LIN {X 0,Y 115.53,Z 526.027,A -85,B 0,C 180,E1 -30181.612,E2 -30181.612} C_VEL
LIN {X 0,Y 120.51,Z 530.093,A -85,B 0,C 180,E1 -30175.516,E2 -30175.516} C_VEL
LIN {X 0,Y 127.732,Z 533.715,A -85,B 0,C 180,E1 -30169.276,E2 -30169.276} C_VEL
LIN {X 0,Y 137.279,Z 536.546,A -85,B 0,C 180,E1 -30163.425,E2 -30163.425} C_VEL
LIN {X 0,Y 149.17,Z 538.493,A -85,B 0,C 180,E1 -30158.125,E2 -30158.125} C_VEL
LIN {X 0,Y 161.998,Z 539.441,A -85,B 0,C 180,E1 -30153.813,E2 -30153.813} C_VEL
LIN {X 0,Y 176.224,Z 539.515,A -85,B 0,C 180,E1 -30150,E2 -30150} C_VEL
LIN {X 0,Y 161.998,Z 539.441,A -85,B 0,C 180,E1 -30146.187,E2 -30146.187} C_VEL
LIN {X 0,Y 156.307,Z 539.2,A -85,B 0,C 180,E1 -30144.414,E2 -30144.414} C_VEL
LIN {X 0,Y 151.525,Z 539.005,A -85,B 0,C 180,E1 -30143.113,E2 -30143.113} C_VEL
LIN {X 0,Y 135.833,Z 538.437,A -85,B 0,C 180,E1 -30139.705,E2 -30139.705} C_VEL
LIN {X 0,Y 131.312,Z 537.898,A -85,B 0,C 180,E1 -30138.103,E2 -30138.103} C_VEL
LIN {X 0,Y 130.038,Z 537.644,A -85,B 0,C 180,E1 -30137.459,E2 -30137.459} C_VEL
LIN {X 0,Y 123.595,Z 536.121,A -85,B 0,C 180,E1 -30133.482,E2 -30133.482} C_VEL
LIN {X 0,Y 115.033,Z 532.752,A -85,B 0,C 180,E1 -30126.405,E2 -30126.405} C_VEL
LIN {X 0,Y 108.205,Z 527.615,A -85,B 0,C 180,E1 -30117.599,E2 -30117.599} C_VEL
LIN {X 0,Y 105.051,Z 522.639,A -85,B 0,C 180,E1 -30110.293,E2 -30110.293} C_VEL
LIN {X 0,Y 103.843,Z 517.611,A -85,B 0,C 180,E1 -30103.904,E2 -30103.904} C_VEL
LIN {X 0,Y 104.036,Z 511.583,A -85,B 0,C 180,E1 -30097.441,E2 -30097.441} C_VEL
LIN {X 0,Y 105.392,Z 504.732,A -85,B 0,C 180,E1 -30091.29,E2 -30091.29} C_VEL
LIN {X 0,Y 107.89,Z 496.243,A -85,B 0,C 180,E1 -30085.046,E2 -30085.046} C_VEL
LIN {X 0,Y 110.837,Z 487.656,A -85,B 0,C 180,E1 -30079.923,E2 -30079.923} C_VEL
LIN {X 0,Y 114.109,Z 478.288,A -85,B 0,C 180,E1 -30075.415,E2 -30075.415} C_VEL
LIN {X 0,Y 115.916,Z 472.807,A -85,B 0,C 180,E1 -30072.918,E2 -30072.918} C_VEL
LIN {X 0,Y 116.839,Z 468.521,A -85,B 0,C 180,E1 -30070.394,E2 -30070.394} C_VEL
LIN {X 0,Y 117.39,Z 465.488,A -85,B 0,C 180,E1 -30067.787,E2 -30067.787} C_VEL
LIN {X 0,Y 117.568,Z 464.579,A -85,B 0,C 180,E1 -30066.865,E2 -30066.865} C_VEL
LIN {X 0,Y 117.839,Z 462.307,A -85,B 0,C 180,E1 -30063.417,E2 -30063.417} C_VEL
LIN {X 0,Y 118.156,Z 460.957,A -85,B 0,C 180,E1 -30059.998,E2 -30059.998} C_VEL
LIN {X 0,Y 117.866,Z 461.826,A -85,B 0,C 180,E1 -30059.712,E2 -30059.712} C_VEL
LIN {X 0,Y 112.451,Z 474.621,A -85,B 0,C 180,E1 -30059.431,E2 -30059.431} C_VEL
LIN {X 0,Y 106.309,Z 485.523,A -85,B 0,C 180,E1 -30059.086,E2 -30059.086} C_VEL
LIN {X 0,Y 100.172,Z 494.46,A -85,B 0,C 180,E1 -30058.699,E2 -30058.699} C_VEL
LIN {X 0,Y 93.165,Z 502.98,A -85,B 0,C 180,E1 -30058.202,E2 -30058.202} C_VEL
LIN {X 0,Y 86.169,Z 510.193,A -85,B 0,C 180,E1 -30057.561,E2 -30057.561} C_VEL
LIN {X 0,Y 79.184,Z 516.388,A -85,B 0,C 180,E1 -30056.836,E2 -30056.836} C_VEL
LIN {X 0,Y 70.48,Z 522.921,A -85,B 0,C 180,E1 -30055.659,E2 -30055.659} C_VEL
LIN {X 0,Y 61.651,Z 528.476,A -85,B 0,C 180,E1 -30054.038,E2 -30054.038} C_VEL
LIN {X 0,Y 52.375,Z 533.31,A -85,B 0,C 180,E1 -30051.657,E2 -30051.657} C_VEL
LIN {X 0,Y 43.038,Z 537.243,A -85,B 0,C 180,E1 -30048.451,E2 -30048.451} C_VEL
LIN {X 0,Y 36.381,Z 539.615,A -85,B 0,C 180,E1 -30044.987,E2 -30044.987} C_VEL
LIN {X 0,Y 29.882,Z 541.418,A -85,B 0,C 180,E1 -30040.178,E2 -30040.178} C_VEL
LIN {X 0,Y 18.304,Z 543.885,A -85,B 0,C 180,E1 -30020.164,E2 -30020.164} C_VEL
LIN {X 0,Y 14.225,Z 544.486,A -85,B 0,C 180,E1 -29999.608,E2 -29999.608} C_VEL
LIN {X 0,Y 12.872,Z 544.652,A -85,B 0,C 180,E1 -29970,E2 -29970} C_VEL
LIN {X 0,Y 14.256,Z 544.487,A -85,B 0,C 180,E1 -29940.464,E2 -29940.464} C_VEL
LIN {X 0,Y 18.309,Z 543.885,A -85,B 0,C 180,E1 -29919.854,E2 -29919.854} C_VEL
LIN {X 0,Y 29.882,Z 541.418,A -85,B 0,C 180,E1 -29899.823,E2 -29899.823} C_VEL
LIN {X 0,Y 39.699,Z 538.463,A -85,B 0,C 180,E1 -29893.184,E2 -29893.184} C_VEL
LIN {X 0,Y 49.826,Z 534.472,A -85,B 0,C 180,E1 -29889.129,E2 -29889.129} C_VEL
LIN {X 0,Y 56.656,Z 531.254,A -85,B 0,C 180,E1 -29887.088,E2 -29887.088} C_VEL
LIN {X 0,Y 67.008,Z 525.231,A -85,B 0,C 180,E1 -29884.883,E2 -29884.883} C_VEL
LIN {X 0,Y 75.698,Z 519.138,A -85,B 0,C 180,E1 -29883.592,E2 -29883.592} C_VEL
LIN {X 0,Y 84.419,Z 511.817,A -85,B 0,C 180,E1 -29882.578,E2 -29882.578} C_VEL
LIN {X 0,Y 91.412,Z 504.896,A -85,B 0,C 180,E1 -29881.903,E2 -29881.903} C_VEL
LIN {X 0,Y 98.419,Z 496.726,A -85,B 0,C 180,E1 -29881.402,E2 -29881.402} C_VEL
LIN {X 0,Y 104.555,Z 488.223,A -85,B 0,C 180,E1 -29881.004,E2 -29881.004} C_VEL
LIN {X 0,Y 109.818,Z 479.515,A -85,B 0,C 180,E1 -29880.71,E2 -29880.71} C_VEL
LIN {X 0,Y 114.593,Z 469.885,A -85,B 0,C 180,E1 -29880.479,E2 -29880.479} C_VEL
LIN {X 0,Y 117.865,Z 461.832,A -85,B 0,C 180,E1 -29880.325,E2 -29880.325} C_VEL
LIN {X 0,Y 118.162,Z 460.939,A -85,B 0,C 180,E1 -29880.002,E2 -29880.002} C_VEL
LIN {X 0,Y 117.775,Z 462.852,A -85,B 0,C 180,E1 -29875.578,E2 -29875.578} C_VEL
LIN {X 0,Y 117.585,Z 464.537,A -85,B 0,C 180,E1 -29873.136,E2 -29873.136} C_VEL
LIN {X 0,Y 117.066,Z 467.337,A -85,B 0,C 180,E1 -29870.499,E2 -29870.499} C_VEL
LIN {X 0,Y 116.536,Z 470.027,A -85,B 0,C 180,E1 -29868.611,E2 -29868.611} C_VEL
LIN {X 0,Y 115.614,Z 473.856,A -85,B 0,C 180,E1 -29866.554,E2 -29866.554} C_VEL
LIN {X 0,Y 111.97,Z 484.489,A -85,B 0,C 180,E1 -29861.712,E2 -29861.712} C_VEL
LIN {X 0,Y 109.139,Z 492.578,A -85,B 0,C 180,E1 -29857.273,E2 -29857.273} C_VEL
LIN {X 0,Y 106.805,Z 499.724,A -85,B 0,C 180,E1 -29852.576,E2 -29852.576} C_VEL
LIN {X 0,Y 104.762,Z 507.268,A -85,B 0,C 180,E1 -29846.586,E2 -29846.586} C_VEL
LIN {X 0,Y 103.737,Z 514.599,A -85,B 0,C 180,E1 -29839.467,E2 -29839.467} C_VEL
LIN {X 0,Y 104.4,Z 520.737,A -85,B 0,C 180,E1 -29832.229,E2 -29832.229} C_VEL
LIN {X 0,Y 106.954,Z 526.067,A -85,B 0,C 180,E1 -29824.784,E2 -29824.784} C_VEL
LIN {X 0,Y 111.232,Z 530.386,A -85,B 0,C 180,E1 -29817.806,E2 -29817.806} C_VEL
LIN {X 0,Y 117.751,Z 534.005,A -85,B 0,C 180,E1 -29810.984,E2 -29810.984} C_VEL
LIN {X 0,Y 124.29,Z 536.317,A -85,B 0,C 180,E1 -29806.005,E2 -29806.005} C_VEL
LIN {X 0,Y 135.51,Z 538.538,A -85,B 0,C 180,E1 -29799.812,E2 -29799.812} C_VEL
LIN {X 0,Y 148.1,Z 539.687,A -85,B 0,C 180,E1 -29794.785,E2 -29794.785} C_VEL
LIN {X 0,Y 164.311,Z 539.834,A -85,B 0,C 180,E1 -29790,E2 -29790} C_VEL
LIN {X 0,Y 148.1,Z 539.687,A -85,B 0,C 180,E1 -29785.215,E2 -29785.215} C_VEL
LIN {X 0,Y 135.51,Z 538.538,A -85,B 0,C 180,E1 -29780.188,E2 -29780.188} C_VEL
LIN {X 0,Y 130.038,Z 537.644,A -85,B 0,C 180,E1 -29777.459,E2 -29777.459} C_VEL
LIN {X 0,Y 125.995,Z 536.984,A -85,B 0,C 180,E1 -29775.552,E2 -29775.552} C_VEL
LIN {X 0,Y 112.333,Z 535.461,A -85,B 0,C 180,E1 -29770.066,E2 -29770.066} C_VEL
LIN {X 0,Y 108.732,Z 534.57,A -85,B 0,C 180,E1 -29767.694,E2 -29767.694} C_VEL
LIN {X 0,Y 107.819,Z 534.193,A -85,B 0,C 180,E1 -29766.796,E2 -29766.796} C_VEL
LIN {X 0,Y 102.19,Z 530.522,A -85,B 0,C 180,E1 -29759.259,E2 -29759.259} C_VEL
LIN {X 0,Y 98.44,Z 525.194,A -85,B 0,C 180,E1 -29750.02,E2 -29750.02} C_VEL
LIN {X 0,Y 97.559,Z 518.271,A -85,B 0,C 180,E1 -29740.414,E2 -29740.414} C_VEL
LIN {X 0,Y 98.89,Z 511.152,A -85,B 0,C 180,E1 -29732.537,E2 -29732.537} C_VEL
LIN {X 0,Y 101.524,Z 503.604,A -85,B 0,C 180,E1 -29725.854,E2 -29725.854} C_VEL
LIN {X 0,Y 104.848,Z 495.671,A -85,B 0,C 180,E1 -29720.215,E2 -29720.215} C_VEL
LIN {X 0,Y 108.168,Z 488.054,A -85,B 0,C 180,E1 -29715.776,E2 -29715.776} C_VEL
LIN {X 0,Y 111.823,Z 479.417,A -85,B 0,C 180,E1 -29711.676,E2 -29711.676} C_VEL
LIN {X 0,Y 113.231,Z 475.646,A -85,B 0,C 180,E1 -29709.754,E2 -29709.754} C_VEL
LIN {X 0,Y 114.361,Z 471.98,A -85,B 0,C 180,E1 -29707.058,E2 -29707.058} C_VEL
LIN {X 0,Y 114.739,Z 470.338,A -85,B 0,C 180,E1 -29705.27,E2 -29705.27} C_VEL
LIN {X 0,Y 115.032,Z 469.144,A -85,B 0,C 180,E1 -29703.501,E2 -29703.501} C_VEL
LIN {X 0,Y 114.177,Z 471.006,A -85,B 0,C 180,E1 -29703.048,E2 -29703.048} C_VEL
LIN {X 0,Y 108.194,Z 482.562,A -85,B 0,C 180,E1 -29702.924,E2 -29702.924} C_VEL
LIN {X 0,Y 101.146,Z 493.131,A -85,B 0,C 180,E1 -29702.797,E2 -29702.797} C_VEL
LIN {X 0,Y 94.976,Z 500.868,A -85,B 0,C 180,E1 -29702.633,E2 -29702.633} C_VEL
LIN {X 0,Y 86.16,Z 509.999,A -85,B 0,C 180,E1 -29702.297,E2 -29702.297} C_VEL
LIN {X 0,Y 79.111,Z 516.194,A -85,B 0,C 180,E1 -29701.987,E2 -29701.987} C_VEL
LIN {X 0,Y 70.301,Z 522.727,A -85,B 0,C 180,E1 -29701.455,E2 -29701.455} C_VEL
LIN {X 0,Y 63.258,Z 527.227,A -85,B 0,C 180,E1 -29700.888,E2 -29700.888} C_VEL
LIN {X 0,Y 53.476,Z 532.382,A -85,B 0,C 180,E1 -29699.749,E2 -29699.749} C_VEL
LIN {X 0,Y 45.696,Z 535.808,A -85,B 0,C 180,E1 -29698.546,E2 -29698.546} C_VEL
LIN {X 0,Y 35.215,Z 539.42,A -85,B 0,C 180,E1 -29696.245,E2 -29696.245} C_VEL
LIN {X 0,Y 28.272,Z 541.223,A -85,B 0,C 180,E1 -29693.889,E2 -29693.889} C_VEL
LIN {X 0,Y 14.789,Z 543.69,A -85,B 0,C 180,E1 -29681.885,E2 -29681.885} C_VEL
LIN {X 0,Y 8.78,Z 544.292,A -85,B 0,C 180,E1 -29663.168,E2 -29663.168} C_VEL
LIN {X 0,Y 5.758,Z 544.457,A -85,B 0,C 180,E1 -29610,E2 -29610} C_VEL
LIN {X 0,Y 8.798,Z 544.293,A -85,B 0,C 180,E1 -29556.985,E2 -29556.985} C_VEL
LIN {X 0,Y 14.791,Z 543.691,A -85,B 0,C 180,E1 -29538.137,E2 -29538.137} C_VEL
LIN {X 0,Y 28.272,Z 541.223,A -85,B 0,C 180,E1 -29526.112,E2 -29526.112} C_VEL
LIN {X 0,Y 38.7,Z 538.268,A -85,B 0,C 180,E1 -29522.835,E2 -29522.835} C_VEL
LIN {X 0,Y 49.201,Z 534.277,A -85,B 0,C 180,E1 -29520.889,E2 -29520.889} C_VEL
LIN {X 0,Y 56.223,Z 531.059,A -85,B 0,C 180,E1 -29519.85,E2 -29519.85} C_VEL
LIN {X 0,Y 66.779,Z 525.037,A -85,B 0,C 180,E1 -29518.794,E2 -29518.794} C_VEL
LIN {X 0,Y 75.587,Z 518.944,A -85,B 0,C 180,E1 -29518.192,E2 -29518.192} C_VEL
LIN {X 0,Y 84.4,Z 511.622,A -85,B 0,C 180,E1 -29517.738,E2 -29517.738} C_VEL
LIN {X 0,Y 91.452,Z 504.701,A -85,B 0,C 180,E1 -29517.449,E2 -29517.449} C_VEL
LIN {X 0,Y 98.501,Z 496.532,A -85,B 0,C 180,E1 -29517.275,E2 -29517.275} C_VEL
LIN {X 0,Y 104.672,Z 488.029,A -85,B 0,C 180,E1 -29517.113,E2 -29517.113} C_VEL
LIN {X 0,Y 109.959,Z 479.321,A -85,B 0,C 180,E1 -29517.01,E2 -29517.01} C_VEL
LIN {X 0,Y 114.36,Z 470.588,A -85,B 0,C 180,E1 -29516.941,E2 -29516.941} C_VEL
LIN {X 0,Y 115.039,Z 469.127,A -85,B 0,C 180,E1 -29516.499,E2 -29516.499} C_VEL
LIN {X 0,Y 114.766,Z 470.276,A -85,B 0,C 180,E1 -29514.732,E2 -29514.732} C_VEL
LIN {X 0,Y 114.116,Z 472.975,A -85,B 0,C 180,E1 -29512.101,E2 -29512.101} C_VEL
LIN {X 0,Y 113.218,Z 475.674,A -85,B 0,C 180,E1 -29510.238,E2 -29510.238} C_VEL
LIN {X 0,Y 111.827,Z 479.404,A -85,B 0,C 180,E1 -29508.331,E2 -29508.331} C_VEL
LIN {X 0,Y 107.548,Z 489.598,A -85,B 0,C 180,E1 -29503.396,E2 -29503.396} C_VEL
LIN {X 0,Y 103.013,Z 500.012,A -85,B 0,C 180,E1 -29496.906,E2 -29496.906} C_VEL
LIN {X 0,Y 99.623,Z 508.727,A -85,B 0,C 180,E1 -29489.784,E2 -29489.784} C_VEL
LIN {X 0,Y 97.978,Z 514.853,A -85,B 0,C 180,E1 -29483.581,E2 -29483.581} C_VEL
LIN {X 0,Y 97.475,Z 520.931,A -85,B 0,C 180,E1 -29476.136,E2 -29476.136} C_VEL
LIN {X 0,Y 98.796,Z 526.081,A -85,B 0,C 180,E1 -29468.513,E2 -29468.513} C_VEL
LIN {X 0,Y 102.139,Z 530.53,A -85,B 0,C 180,E1 -29460.749,E2 -29460.749} C_VEL
LIN {X 0,Y 108.005,Z 534.292,A -85,B 0,C 180,E1 -29452.98,E2 -29452.98} C_VEL
LIN {X 0,Y 113.262,Z 536.417,A -85,B 0,C 180,E1 -29448.074,E2 -29448.074} C_VEL
LIN {X 0,Y 122.132,Z 538.533,A -85,B 0,C 180,E1 -29441.981,E2 -29441.981} C_VEL
LIN {X 0,Y 134.521,Z 539.916,A -85,B 0,C 180,E1 -29435.998,E2 -29435.998} C_VEL
LIN {X 0,Y 147.626,Z 540.282,A -85,B 0,C 180,E1 -29431.378,E2 -29431.378} C_VEL
LIN {X 0,Y 152.405,Z 540.153,A -85,B 0,C 180,E1 -29430,E2 -29430} C_VEL
LIN {X 0,Y 140.832,Z 540.169,A -85,B 0,C 180,E1 -29426.413,E2 -29426.413} C_VEL
LIN {X 0,Y 128.022,Z 539.297,A -85,B 0,C 180,E1 -29421.157,E2 -29421.157} C_VEL
LIN {X 0,Y 119.45,Z 537.971,A -85,B 0,C 180,E1 -29416.388,E2 -29416.388} C_VEL
LIN {X 0,Y 111.734,Z 535.891,A -85,B 0,C 180,E1 -29410.64,E2 -29410.64} C_VEL
LIN {X 0,Y 107.819,Z 534.193,A -85,B 0,C 180,E1 -29406.796,E2 -29406.796} C_VEL
LIN {X 0,Y 104.89,Z 533.159,A -85,B 0,C 180,E1 -29404.087,E2 -29404.087} C_VEL
LIN {X 0,Y 94.721,Z 530.474,A -85,B 0,C 180,E1 -29395.798,E2 -29395.798} C_VEL
LIN {X 0,Y 92.539,Z 529.043,A -85,B 0,C 180,E1 -29392.569,E2 -29392.569} C_VEL
LIN {X 0,Y 92.134,Z 528.439,A -85,B 0,C 180,E1 -29391.437,E2 -29391.437} C_VEL
LIN {X 0,Y 91.087,Z 524.144,A -85,B 0,C 180,E1 -29383.977,E2 -29383.977} C_VEL
LIN {X 0,Y 91.954,Z 517.723,A -85,B 0,C 180,E1 -29374.969,E2 -29374.969} C_VEL
LIN {X 0,Y 94.409,Z 511.216,A -85,B 0,C 180,E1 -29367.722,E2 -29367.722} C_VEL
LIN {X 0,Y 97.995,Z 503.845,A -85,B 0,C 180,E1 -29361.202,E2 -29361.202} C_VEL
LIN {X 0,Y 102.179,Z 495.907,A -85,B 0,C 180,E1 -29355.654,E2 -29355.654} C_VEL
LIN {X 0,Y 106.153,Z 488.365,A -85,B 0,C 180,E1 -29351.454,E2 -29351.454} C_VEL
LIN {X 0,Y 109.817,Z 480.976,A -85,B 0,C 180,E1 -29347.881,E2 -29347.881} C_VEL
LIN {X 0,Y 110.214,Z 480.011,A -85,B 0,C 180,E1 -29347.325,E2 -29347.325} C_VEL
LIN {X 0,Y 109.156,Z 481.709,A -85,B 0,C 180,E1 -29346.66,E2 -29346.66} C_VEL
LIN {X 0,Y 101.739,Z 492.937,A -85,B 0,C 180,E1 -29346.793,E2 -29346.793} C_VEL
LIN {X 0,Y 95.565,Z 500.675,A -85,B 0,C 180,E1 -29346.885,E2 -29346.885} C_VEL
LIN {X 0,Y 86.738,Z 509.804,A -85,B 0,C 180,E1 -29347.004,E2 -29347.004} C_VEL
LIN {X 0,Y 79.677,Z 515.999,A -85,B 0,C 180,E1 -29347.118,E2 -29347.118} C_VEL
LIN {X 0,Y 70.843,Z 522.532,A -85,B 0,C 180,E1 -29347.237,E2 -29347.237} C_VEL
LIN {X 0,Y 63.769,Z 527.032,A -85,B 0,C 180,E1 -29347.31,E2 -29347.31} C_VEL
LIN {X 0,Y 52.924,Z 532.625,A -85,B 0,C 180,E1 -29347.375,E2 -29347.375} C_VEL
LIN {X 0,Y 42.541,Z 536.854,A -85,B 0,C 180,E1 -29347.601,E2 -29347.601} C_VEL
LIN {X 0,Y 35.467,Z 539.226,A -85,B 0,C 180,E1 -29347.798,E2 -29347.798} C_VEL
LIN {X 0,Y 28.41,Z 541.029,A -85,B 0,C 180,E1 -29348.313,E2 -29348.313} C_VEL
LIN {X 0,Y 14.284,Z 543.495,A -85,B 0,C 180,E1 -29350.265,E2 -29350.265} C_VEL
LIN {X 0,Y 7.271,Z 544.097,A -85,B 0,C 180,E1 -29354.864,E2 -29354.864} C_VEL
LIN {X 0,Y 1.342,Z 544.264,A -85,B 0,C 180,E1 -29430,E2 -29430} C_VEL
LIN {X 0,Y 7.264,Z 544.098,A -85,B 0,C 180,E1 -29505.336,E2 -29505.336} C_VEL
LIN {X 0,Y 14.283,Z 543.496,A -85,B 0,C 180,E1 -29509.757,E2 -29509.757} C_VEL
LIN {X 0,Y 28.41,Z 541.029,A -85,B 0,C 180,E1 -29511.687,E2 -29511.687} C_VEL
LIN {X 0,Y 39.006,Z 538.072,A -85,B 0,C 180,E1 -29512.286,E2 -29512.286} C_VEL
LIN {X 0,Y 49.607,Z 534.082,A -85,B 0,C 180,E1 -29512.609,E2 -29512.609} C_VEL
LIN {X 0,Y 60.238,Z 528.947,A -85,B 0,C 180,E1 -29512.604,E2 -29512.604} C_VEL
LIN {X 0,Y 69.074,Z 523.687,A -85,B 0,C 180,E1 -29512.749,E2 -29512.749} C_VEL
LIN {X 0,Y 77.911,Z 517.374,A -85,B 0,C 180,E1 -29512.853,E2 -29512.853} C_VEL
LIN {X 0,Y 84.979,Z 511.428,A -85,B 0,C 180,E1 -29512.934,E2 -29512.934} C_VEL
LIN {X 0,Y 92.043,Z 504.507,A -85,B 0,C 180,E1 -29513.026,E2 -29513.026} C_VEL
LIN {X 0,Y 99.092,Z 496.338,A -85,B 0,C 180,E1 -29513.173,E2 -29513.173} C_VEL
LIN {X 0,Y 105.269,Z 487.835,A -85,B 0,C 180,E1 -29513.25,E2 -29513.25} C_VEL
LIN {X 0,Y 109.166,Z 481.695,A -85,B 0,C 180,E1 -29513.327,E2 -29513.327} C_VEL
LIN {X 0,Y 110.222,Z 479.996,A -85,B 0,C 180,E1 -29512.676,E2 -29512.676} C_VEL
LIN {X 0,Y 108.059,Z 484.613,A -85,B 0,C 180,E1 -29510.371,E2 -29510.371} C_VEL
LIN {X 0,Y 103.854,Z 492.82,A -85,B 0,C 180,E1 -29506.176,E2 -29506.176} C_VEL
LIN {X 0,Y 99.128,Z 501.682,A -85,B 0,C 180,E1 -29500.436,E2 -29500.436} C_VEL
LIN {X 0,Y 95.443,Z 508.971,A -85,B 0,C 180,E1 -29494.419,E2 -29494.419} C_VEL
LIN {X 0,Y 92.738,Z 515.274,A -85,B 0,C 180,E1 -29487.965,E2 -29487.965} C_VEL
LIN {X 0,Y 91.17,Z 521.19,A -85,B 0,C 180,E1 -29480.43,E2 -29480.43} C_VEL
LIN {X 0,Y 91.33,Z 526.254,A -85,B 0,C 180,E1 -29472.501,E2 -29472.501} C_VEL
LIN {X 0,Y 93.531,Z 530.627,A -85,B 0,C 180,E1 -29464.258,E2 -29464.258} C_VEL
LIN {X 0,Y 98.459,Z 534.578,A -85,B 0,C 180,E1 -29455.358,E2 -29455.358} C_VEL
LIN {X 0,Y 104.092,Z 536.965,A -85,B 0,C 180,E1 -29449.057,E2 -29449.057} C_VEL
LIN {X 0,Y 114.583,Z 539.286,A -85,B 0,C 180,E1 -29441.088,E2 -29441.088} C_VEL
LIN {X 0,Y 123.077,Z 540.226,A -85,B 0,C 180,E1 -29436.558,E2 -29436.558} C_VEL
LIN {X 0,Y 133.634,Z 540.627,A -85,B 0,C 180,E1 -29432.281,E2 -29432.281} C_VEL
LIN {X 0,Y 140.49,Z 540.472,A -85,B 0,C 180,E1 -29430,E2 -29430} C_VEL
LIN {X 0,Y 131.511,Z 540.565,A -85,B 0,C 180,E1 -29426.937,E2 -29426.937} C_VEL
LIN {X 0,Y 120.584,Z 540.045,A -85,B 0,C 180,E1 -29422.211,E2 -29422.211} C_VEL
LIN {X 0,Y 108.962,Z 538.266,A -85,B 0,C 180,E1 -29415.049,E2 -29415.049} C_VEL
LIN {X 0,Y 101.541,Z 535.979,A -85,B 0,C 180,E1 -29408.287,E2 -29408.287} C_VEL
LIN {X 0,Y 94.891,Z 532.04,A -85,B 0,C 180,E1 -29398.773,E2 -29398.773} C_VEL
LIN {X 0,Y 92.134,Z 528.439,A -85,B 0,C 180,E1 -29391.437,E2 -29391.437} C_VEL
LIN {X 0,Y 90.803,Z 526.757,A -85,B 0,C 180,E1 -29387.988,E2 -29387.988} C_VEL
LIN {X 0,Y 86.123,Z 522.502,A -85,B 0,C 180,E1 -29377.176,E2 -29377.176} C_VEL
LIN {X 0,Y 85.979,Z 520.542,A -85,B 0,C 180,E1 -29373.482,E2 -29373.482} C_VEL
LIN {X 0,Y 86.244,Z 519.758,A -85,B 0,C 180,E1 -29372.297,E2 -29372.297} C_VEL
LIN {X 0,Y 89.862,Z 512.848,A -85,B 0,C 180,E1 -29364.119,E2 -29364.119} C_VEL
LIN {X 0,Y 94.345,Z 505.462,A -85,B 0,C 180,E1 -29357.333,E2 -29357.333} C_VEL
LIN {X 0,Y 99.444,Z 497.412,A -85,B 0,C 180,E1 -29351.699,E2 -29351.699} C_VEL
LIN {X 0,Y 100.186,Z 496.144,A -85,B 0,C 180,E1 -29350.867,E2 -29350.867} C_VEL
LIN {X 0,Y 93.168,Z 504.314,A -85,B 0,C 180,E1 -29351.302,E2 -29351.302} C_VEL
LIN {X 0,Y 84.371,Z 512.861,A -85,B 0,C 180,E1 -29351.837,E2 -29351.837} C_VEL
LIN {X 0,Y 73.841,Z 521.183,A -85,B 0,C 180,E1 -29352.697,E2 -29352.697} C_VEL
LIN {X 0,Y 65.059,Z 526.838,A -85,B 0,C 180,E1 -29353.54,E2 -29353.54} C_VEL
LIN {X 0,Y 55.435,Z 531.927,A -85,B 0,C 180,E1 -29354.684,E2 -29354.684} C_VEL
LIN {X 0,Y 47.515,Z 535.42,A -85,B 0,C 180,E1 -29355.97,E2 -29355.97} C_VEL
LIN {X 0,Y 37.116,Z 539.031,A -85,B 0,C 180,E1 -29358.783,E2 -29358.783} C_VEL
LIN {X 0,Y 23.544,Z 542.23,A -85,B 0,C 180,E1 -29366.427,E2 -29366.427} C_VEL
LIN {X 0,Y 17.068,Z 543.301,A -85,B 0,C 180,E1 -29374.56,E2 -29374.56} C_VEL
LIN {X 0,Y 11.406,Z 543.903,A -85,B 0,C 180,E1 -29391.966,E2 -29391.966} C_VEL
LIN {X 0,Y 8.433,Z 544.07,A -85,B 0,C 180,E1 -29430,E2 -29430} C_VEL
LIN {X 0,Y 11.389,Z 543.903,A -85,B 0,C 180,E1 -29468.101,E2 -29468.101} C_VEL
LIN {X 0,Y 17.065,Z 543.301,A -85,B 0,C 180,E1 -29485.452,E2 -29485.452} C_VEL
LIN {X 0,Y 30.268,Z 540.835,A -85,B 0,C 180,E1 -29498.242,E2 -29498.242} C_VEL
LIN {X 0,Y 40.587,Z 537.877,A -85,B 0,C 180,E1 -29502.242,E2 -29502.242} C_VEL
LIN {X 0,Y 47.518,Z 535.419,A -85,B 0,C 180,E1 -29504.016,E2 -29504.016} C_VEL
LIN {X 0,Y 58.043,Z 530.669,A -85,B 0,C 180,E1 -29505.612,E2 -29505.612} C_VEL
LIN {X 0,Y 68.572,Z 524.648,A -85,B 0,C 180,E1 -29506.816,E2 -29506.816} C_VEL
LIN {X 0,Y 77.355,Z 518.555,A -85,B 0,C 180,E1 -29507.595,E2 -29507.595} C_VEL
LIN {X 0,Y 84.384,Z 512.859,A -85,B 0,C 180,E1 -29508.121,E2 -29508.121} C_VEL
LIN {X 0,Y 93.172,Z 504.314,A -85,B 0,C 180,E1 -29508.688,E2 -29508.688} C_VEL
LIN {X 0,Y 100.183,Z 496.145,A -85,B 0,C 180,E1 -29509.142,E2 -29509.142} C_VEL
LIN {X 0,Y 94.35,Z 505.456,A -85,B 0,C 180,E1 -29502.668,E2 -29502.668} C_VEL
LIN {X 0,Y 89.038,Z 514.197,A -85,B 0,C 180,E1 -29494.522,E2 -29494.522} C_VEL
LIN {X 0,Y 85.528,Z 521.444,A -85,B 0,C 180,E1 -29485.255,E2 -29485.255} C_VEL
LIN {X 0,Y 84.543,Z 525.778,A -85,B 0,C 180,E1 -29478.318,E2 -29478.318} C_VEL
LIN {X 0,Y 85.383,Z 530.66,A -85,B 0,C 180,E1 -29468.568,E2 -29468.568} C_VEL
LIN {X 0,Y 89.317,Z 534.857,A -85,B 0,C 180,E1 -29458.171,E2 -29458.171} C_VEL
LIN {X 0,Y 93.455,Z 536.993,A -85,B 0,C 180,E1 -29452.086,E2 -29452.086} C_VEL
LIN {X 0,Y 101.464,Z 539.209,A -85,B 0,C 180,E1 -29444.145,E2 -29444.145} C_VEL
LIN {X 0,Y 113.189,Z 540.585,A -85,B 0,C 180,E1 -29436.579,E2 -29436.579} C_VEL
LIN {X 0,Y 126.513,Z 540.847,A -85,B 0,C 180,E1 -29430.819,E2 -29430.819} C_VEL
LIN {X 0,Y 128.847,Z 540.784,A -85,B 0,C 180,E1 -29430,E2 -29430} C_VEL
LIN {X 0,Y 119.694,Z 540.864,A -85,B 0,C 180,E1 -29426.511,E2 -29426.511} C_VEL
LIN {X 0,Y 107.081,Z 540.017,A -85,B 0,C 180,E1 -29419.881,E2 -29419.881} C_VEL
LIN {X 0,Y 98.692,Z 538.557,A -85,B 0,C 180,E1 -29413.451,E2 -29413.451} C_VEL
LIN {X 0,Y 92.191,Z 536.396,A -85,B 0,C 180,E1 -29406.171,E2 -29406.171} C_VEL
LIN {X 0,Y 86.478,Z 532.314,A -85,B 0,C 180,E1 -29395.329,E2 -29395.329} C_VEL
LIN {X 0,Y 84.543,Z 527.478,A -85,B 0,C 180,E1 -29384.955,E2 -29384.955} C_VEL
LIN {X 0,Y 85.554,Z 521.443,A -85,B 0,C 180,E1 -29374.77,E2 -29374.77} C_VEL
LIN {X 0,Y 86.244,Z 519.758,A -85,B 0,C 180,E1 -29372.297,E2 -29372.297} C_VEL
LIN {X 0,Y 86.504,Z 518.36,A -85,B 0,C 180,E1 -29369.819,E2 -29369.819} C_VEL
LIN {X 0,Y 85.647,Z 514.934,A -85,B 0,C 180,E1 -29361.146,E2 -29361.146} C_VEL
LIN {X 0,Y 86.48,Z 513.232,A -85,B 0,C 180,E1 -29358.816,E2 -29358.816} C_VEL
LIN {X 0,Y 88.038,Z 511.023,A -85,B 0,C 180,E1 -29356.68,E2 -29356.68} C_VEL
LIN {X 0,Y 87.861,Z 511.04,A -85,B 0,C 180,E1 -29356.289,E2 -29356.289} C_VEL
LIN {X 0,Y 80.923,Z 516.986,A -85,B 0,C 180,E1 -29357.196,E2 -29357.196} C_VEL
LIN {X 0,Y 72.271,Z 523.298,A -85,B 0,C 180,E1 -29358.537,E2 -29358.537} C_VEL
LIN {X 0,Y 63.64,Z 528.559,A -85,B 0,C 180,E1 -29360.171,E2 -29360.171} C_VEL
LIN {X 0,Y 53.357,Z 533.692,A -85,B 0,C 180,E1 -29362.78,E2 -29362.78} C_VEL
LIN {X 0,Y 43.299,Z 537.683,A -85,B 0,C 180,E1 -29366.784,E2 -29366.784} C_VEL
LIN {X 0,Y 33.56,Z 540.64,A -85,B 0,C 180,E1 -29373.107,E2 -29373.107} C_VEL
LIN {X 0,Y 21.912,Z 543.106,A -85,B 0,C 180,E1 -29390.1,E2 -29390.1} C_VEL
LIN {X 0,Y 17.562,Z 543.708,A -85,B 0,C 180,E1 -29406.411,E2 -29406.411} C_VEL
LIN {X 0,Y 15.543,Z 543.876,A -85,B 0,C 180,E1 -29430,E2 -29430} C_VEL
LIN {X 0,Y 17.546,Z 543.709,A -85,B 0,C 180,E1 -29453.612,E2 -29453.612} C_VEL
LIN {X 0,Y 21.909,Z 543.106,A -85,B 0,C 180,E1 -29469.906,E2 -29469.906} C_VEL
LIN {X 0,Y 33.56,Z 540.64,A -85,B 0,C 180,E1 -29486.893,E2 -29486.893} C_VEL
LIN {X 0,Y 43.299,Z 537.682,A -85,B 0,C 180,E1 -29493.214,E2 -29493.214} C_VEL
LIN {X 0,Y 53.37,Z 533.691,A -85,B 0,C 180,E1 -29497.185,E2 -29497.185} C_VEL
LIN {X 0,Y 63.662,Z 528.557,A -85,B 0,C 180,E1 -29499.774,E2 -29499.774} C_VEL
LIN {X 0,Y 72.271,Z 523.298,A -85,B 0,C 180,E1 -29501.463,E2 -29501.463} C_VEL
LIN {X 0,Y 80.924,Z 516.986,A -85,B 0,C 180,E1 -29502.802,E2 -29502.802} C_VEL
LIN {X 0,Y 87.87,Z 511.04,A -85,B 0,C 180,E1 -29503.69,E2 -29503.69} C_VEL
LIN {X 0,Y 88.029,Z 511.024,A -85,B 0,C 180,E1 -29503.341,E2 -29503.341} C_VEL
LIN {X 0,Y 82.509,Z 518.748,A -85,B 0,C 180,E1 -29494.796,E2 -29494.796} C_VEL
LIN {X 0,Y 78.592,Z 525.98,A -85,B 0,C 180,E1 -29483.591,E2 -29483.591} C_VEL
LIN {X 0,Y 77.931,Z 530.624,A -85,B 0,C 180,E1 -29473.829,E2 -29473.829} C_VEL
LIN {X 0,Y 80.624,Z 535.131,A -85,B 0,C 180,E1 -29461.534,E2 -29461.534} C_VEL
LIN {X 0,Y 84.522,Z 537.492,A -85,B 0,C 180,E1 -29453.851,E2 -29453.851} C_VEL
LIN {X 0,Y 94.36,Z 540.004,A -85,B 0,C 180,E1 -29442.911,E2 -29442.911} C_VEL
LIN {X 0,Y 101.12,Z 540.83,A -85,B 0,C 180,E1 -29437.99,E2 -29437.99} C_VEL
LIN {X 0,Y 112.511,Z 541.23,A -85,B 0,C 180,E1 -29431.978,E2 -29431.978} C_VEL
LIN {X 0,Y 117.33,Z 541.096,A -85,B 0,C 180,E1 -29430,E2 -29430} C_VEL
LIN {X 0,Y 105.857,Z 541.051,A -85,B 0,C 180,E1 -29424.766,E2 -29424.766} C_VEL
LIN {X 0,Y 99.612,Z 540.73,A -85,B 0,C 180,E1 -29421.007,E2 -29421.007} C_VEL
LIN {X 0,Y 88.709,Z 538.843,A -85,B 0,C 180,E1 -29411.525,E2 -29411.525} C_VEL
LIN {X 0,Y 84.099,Z 537.271,A -85,B 0,C 180,E1 -29405.302,E2 -29405.302} C_VEL
LIN {X 0,Y 78.999,Z 533.346,A -85,B 0,C 180,E1 -29393.189,E2 -29393.189} C_VEL
LIN {X 0,Y 77.995,Z 528.409,A -85,B 0,C 180,E1 -29381.382,E2 -29381.382} C_VEL
LIN {X 0,Y 79.749,Z 523.317,A -85,B 0,C 180,E1 -29371.918,E2 -29371.918} C_VEL
LIN {X 0,Y 82.508,Z 518.749,A -85,B 0,C 180,E1 -29365.205,E2 -29365.205} C_VEL
LIN {X 0,Y 86.48,Z 513.232,A -85,B 0,C 180,E1 -29358.816,E2 -29358.816} C_VEL
LIN {X 0,Y 85.976,Z 513.469,A -85,B 0,C 180,E1 -29358.3,E2 -29358.3} C_VEL
LIN {X 0,Y 83.959,Z 514.972,A -85,B 0,C 180,E1 -29358.08,E2 -29358.08} C_VEL
LIN {X 0,Y 80.115,Z 518.157,A -85,B 0,C 180,E1 -29358.889,E2 -29358.889} C_VEL
LIN {X 0,Y 70.926,Z 525.373,A -85,B 0,C 180,E1 -29363.308,E2 -29363.308} C_VEL
LIN {X 0,Y 64.57,Z 529.46,A -85,B 0,C 180,E1 -29366.406,E2 -29366.406} C_VEL
LIN {X 0,Y 62.262,Z 530.713,A -85,B 0,C 180,E1 -29367.276,E2 -29367.276} C_VEL
LIN {X 0,Y 53.246,Z 535.03,A -85,B 0,C 180,E1 -29370.915,E2 -29370.915} C_VEL
LIN {X 0,Y 43.861,Z 538.641,A -85,B 0,C 180,E1 -29376.759,E2 -29376.759} C_VEL
LIN {X 0,Y 37.933,Z 540.445,A -85,B 0,C 180,E1 -29382.177,E2 -29382.177} C_VEL
LIN {X 0,Y 27.754,Z 542.911,A -85,B 0,C 180,E1 -29399.573,E2 -29399.573} C_VEL
LIN {X 0,Y 24.268,Z 543.514,A -85,B 0,C 180,E1 -29413.167,E2 -29413.167} C_VEL
LIN {X 0,Y 22.642,Z 543.682,A -85,B 0,C 180,E1 -29430,E2 -29430} C_VEL
LIN {X 0,Y 24.254,Z 543.514,A -85,B 0,C 180,E1 -29446.844,E2 -29446.844} C_VEL
LIN {X 0,Y 27.751,Z 542.911,A -85,B 0,C 180,E1 -29460.43,E2 -29460.43} C_VEL
LIN {X 0,Y 37.933,Z 540.445,A -85,B 0,C 180,E1 -29477.823,E2 -29477.823} C_VEL
LIN {X 0,Y 46.943,Z 537.488,A -85,B 0,C 180,E1 -29485.427,E2 -29485.427} C_VEL
LIN {X 0,Y 56.524,Z 533.496,A -85,B 0,C 180,E1 -29490.497,E2 -29490.497} C_VEL
LIN {X 0,Y 66.466,Z 528.363,A -85,B 0,C 180,E1 -29493.994,E2 -29493.994} C_VEL
LIN {X 0,Y 74.837,Z 523.104,A -85,B 0,C 180,E1 -29496.292,E2 -29496.292} C_VEL
LIN {X 0,Y 76.575,Z 521.945,A -85,B 0,C 180,E1 -29496.602,E2 -29496.602} C_VEL
LIN {X 0,Y 72.486,Z 527.747,A -85,B 0,C 180,E1 -29486.313,E2 -29486.313} C_VEL
LIN {X 0,Y 71.149,Z 531.942,A -85,B 0,C 180,E1 -29476.26,E2 -29476.26} C_VEL
LIN {X 0,Y 72.327,Z 535.403,A -85,B 0,C 180,E1 -29465.662,E2 -29465.662} C_VEL
LIN {X 0,Y 74.898,Z 537.551,A -85,B 0,C 180,E1 -29457.98,E2 -29457.98} C_VEL
LIN {X 0,Y 81.196,Z 539.778,A -85,B 0,C 180,E1 -29447.811,E2 -29447.811} C_VEL
LIN {X 0,Y 92.182,Z 541.217,A -85,B 0,C 180,E1 -29437.656,E2 -29437.656} C_VEL
LIN {X 0,Y 98.591,Z 541.52,A -85,B 0,C 180,E1 -29433.677,E2 -29433.677} C_VEL
LIN {X 0,Y 105.989,Z 541.406,A -85,B 0,C 180,E1 -29430,E2 -29430} C_VEL
LIN {X 0,Y 97.814,Z 541.484,A -85,B 0,C 180,E1 -29425.88,E2 -29425.88} C_VEL
LIN {X 0,Y 86.342,Z 540.641,A -85,B 0,C 180,E1 -29417.612,E2 -29417.612} C_VEL
LIN {X 0,Y 78.954,Z 539.126,A -85,B 0,C 180,E1 -29409.143,E2 -29409.143} C_VEL
LIN {X 0,Y 73.756,Z 536.732,A -85,B 0,C 180,E1 -29399.04,E2 -29399.04} C_VEL
LIN {X 0,Y 71.796,Z 534.617,A -85,B 0,C 180,E1 -29391.541,E2 -29391.541} C_VEL
LIN {X 0,Y 71.672,Z 529.849,A -85,B 0,C 180,E1 -29378.331,E2 -29378.331} C_VEL
LIN {X 0,Y 74.857,Z 524.151,A -85,B 0,C 180,E1 -29366.889,E2 -29366.889} C_VEL
LIN {X 0,Y 76.532,Z 521.948,A -85,B 0,C 180,E1 -29363.323,E2 -29363.323} C_VEL
LIN {X 0,Y 69.79,Z 526.448,A -85,B 0,C 180,E1 -29365.001,E2 -29365.001} C_VEL
LIN {X 0,Y 62.262,Z 530.713,A -85,B 0,C 180,E1 -29367.276,E2 -29367.276} C_VEL
LIN {X 0,Y 57.548,Z 533.179,A -85,B 0,C 180,E1 -29369.737,E2 -29369.737} C_VEL
LIN {X 0,Y 50.934,Z 536.673,A -85,B 0,C 180,E1 -29376.639,E2 -29376.639} C_VEL
LIN {X 0,Y 46.286,Z 538.93,A -85,B 0,C 180,E1 -29383.788,E2 -29383.788} C_VEL
LIN {X 0,Y 42.668,Z 540.365,A -85,B 0,C 180,E1 -29389.567,E2 -29389.567} C_VEL
LIN {X 0,Y 41.353,Z 540.72,A -85,B 0,C 180,E1 -29391.499,E2 -29391.499} C_VEL
LIN {X 0,Y 34.099,Z 542.717,A -85,B 0,C 180,E1 -29405.657,E2 -29405.657} C_VEL
LIN {X 0,Y 31.153,Z 543.319,A -85,B 0,C 180,E1 -29416.963,E2 -29416.963} C_VEL
LIN {X 0,Y 29.757,Z 543.488,A -85,B 0,C 180,E1 -29430,E2 -29430} C_VEL
LIN {X 0,Y 31.141,Z 543.32,A -85,B 0,C 180,E1 -29443.043,E2 -29443.043} C_VEL
LIN {X 0,Y 34.096,Z 542.717,A -85,B 0,C 180,E1 -29454.345,E2 -29454.345} C_VEL
LIN {X 0,Y 43.05,Z 540.251,A -85,B 0,C 180,E1 -29470.768,E2 -29470.768} C_VEL
LIN {X 0,Y 51.319,Z 537.293,A -85,B 0,C 180,E1 -29478.867,E2 -29478.867} C_VEL
LIN {X 0,Y 60.362,Z 533.301,A -85,B 0,C 180,E1 -29484.586,E2 -29484.586} C_VEL
LIN {X 0,Y 61.39,Z 532.793,A -85,B 0,C 180,E1 -29485.086,E2 -29485.086} C_VEL
LIN {X 0,Y 65.59,Z 531.015,A -85,B 0,C 180,E1 -29485.854,E2 -29485.854} C_VEL
LIN {X 0,Y 64.408,Z 534.591,A -85,B 0,C 180,E1 -29474.984,E2 -29474.984} C_VEL
LIN {X 0,Y 66.278,Z 537.832,A -85,B 0,C 180,E1 -29461.979,E2 -29461.979} C_VEL
LIN {X 0,Y 69.448,Z 539.407,A -85,B 0,C 180,E1 -29453.877,E2 -29453.877} C_VEL
LIN {X 0,Y 78.815,Z 541.331,A -85,B 0,C 180,E1 -29441.238,E2 -29441.238} C_VEL
LIN {X 0,Y 91.409,Z 541.805,A -85,B 0,C 180,E1 -29431.878,E2 -29431.878} C_VEL
LIN {X 0,Y 94.915,Z 541.708,A -85,B 0,C 180,E1 -29430,E2 -29430} C_VEL
LIN {X 0,Y 84.823,Z 541.672,A -85,B 0,C 180,E1 -29423.829,E2 -29423.829} C_VEL
LIN {X 0,Y 78.823,Z 541.326,A -85,B 0,C 180,E1 -29418.733,E2 -29418.733} C_VEL
LIN {X 0,Y 69.338,Z 539.336,A -85,B 0,C 180,E1 -29405.806,E2 -29405.806} C_VEL
LIN {X 0,Y 65.276,Z 536.825,A -85,B 0,C 180,E1 -29393.846,E2 -29393.846} C_VEL
LIN {X 0,Y 64.621,Z 533.112,A -85,B 0,C 180,E1 -29380.422,E2 -29380.422} C_VEL
LIN {X 0,Y 65.703,Z 530.958,A -85,B 0,C 180,E1 -29374.091,E2 -29374.091} C_VEL
LIN {X 0,Y 61.746,Z 532.603,A -85,B 0,C 180,E1 -29374.683,E2 -29374.683} C_VEL
LIN {X 0,Y 54.22,Z 536.077,A -85,B 0,C 180,E1 -29378.949,E2 -29378.949} C_VEL
LIN {X 0,Y 48.474,Z 538.445,A -85,B 0,C 180,E1 -29383.538,E2 -29383.538} C_VEL
LIN {X 0,Y 41.353,Z 540.72,A -85,B 0,C 180,E1 -29391.499,E2 -29391.499} C_VEL
LIN {X 0,Y 38.003,Z 541.845,A -85,B 0,C 180,E1 -29398.384,E2 -29398.384} C_VEL
LIN {X 0,Y 36.112,Z 542.653,A -85,B 0,C 180,E1 -29407.017,E2 -29407.017} C_VEL
LIN {X 0,Y 36.104,Z 543.317,A -85,B 0,C 180,E1 -29426.081,E2 -29426.081} C_VEL
LIN {X 0,Y 37.71,Z 543.164,A -85,B 0,C 180,E1 -29438.258,E2 -29438.258} C_VEL
LIN {X 0,Y 40.697,Z 542.522,A -85,B 0,C 180,E1 -29450.205,E2 -29450.205} C_VEL
LIN {X 0,Y 48.673,Z 540.056,A -85,B 0,C 180,E1 -29465.279,E2 -29465.279} C_VEL
LIN {X 0,Y 53.64,Z 538.251,A -85,B 0,C 180,E1 -29470.927,E2 -29470.927} C_VEL
LIN {X 0,Y 57.59,Z 536.866,A -85,B 0,C 180,E1 -29472.934,E2 -29472.934} C_VEL
LIN {X 0,Y 60.394,Z 539.681,A -85,B 0,C 180,E1 -29457.741,E2 -29457.741} C_VEL
LIN {X 0,Y 69.708,Z 541.7,A -85,B 0,C 180,E1 -29441.633,E2 -29441.633} C_VEL
LIN {X 0,Y 77.525,Z 542.132,A -85,B 0,C 180,E1 -29434.327,E2 -29434.327} C_VEL
LIN {X 0,Y 83.966,Z 542.007,A -85,B 0,C 180,E1 -29430,E2 -29430} C_VEL
LIN {X 0,Y 76.404,Z 542.07,A -85,B 0,C 180,E1 -29424.722,E2 -29424.722} C_VEL
LIN {X 0,Y 65.986,Z 541.168,A -85,B 0,C 180,E1 -29413.436,E2 -29413.436} C_VEL
LIN {X 0,Y 60.434,Z 539.68,A -85,B 0,C 180,E1 -29402.28,E2 -29402.28} C_VEL
LIN {X 0,Y 57.616,Z 536.853,A -85,B 0,C 180,E1 -29387.038,E2 -29387.038} C_VEL
LIN {X 0,Y 53.639,Z 538.251,A -85,B 0,C 180,E1 -29389.073,E2 -29389.073} C_VEL
LIN {X 0,Y 46.688,Z 540.67,A -85,B 0,C 180,E1 -29397.6,E2 -29397.6} C_VEL
LIN {X 0,Y 40.699,Z 542.522,A -85,B 0,C 180,E1 -29409.796,E2 -29409.796} C_VEL
LIN {X 0,Y 38.118,Z 543.125,A -85,B 0,C 180,E1 -29419.376,E2 -29419.376} C_VEL
LIN {X 0,Y 36.863,Z 543.294,A -85,B 0,C 180,E1 -29430,E2 -29430} C_VEL
LIN {X 0,Y 37.71,Z 543.164,A -85,B 0,C 180,E1 -29438.258,E2 -29438.258} C_VEL
LIN {X 0,Y 39.339,Z 542.981,A -85,B 0,C 180,E1 -29443.576,E2 -29443.576} C_VEL
LIN {X 0,Y 42.005,Z 542.646,A -85,B 0,C 180,E1 -29447.704,E2 -29447.704} C_VEL
LIN {X 0,Y 53.283,Z 540.745,A -85,B 0,C 180,E1 -29456.653,E2 -29456.653} C_VEL
LIN {X 0,Y 59.65,Z 541.982,A -85,B 0,C 180,E1 -29443.629,E2 -29443.629} C_VEL
LIN {X 0,Y 70.325,Z 542.381,A -85,B 0,C 180,E1 -29432.151,E2 -29432.151} C_VEL
LIN {X 0,Y 73.223,Z 542.301,A -85,B 0,C 180,E1 -29430,E2 -29430} C_VEL
LIN {X 0,Y 63.911,Z 542.242,A -85,B 0,C 180,E1 -29421.741,E2 -29421.741} C_VEL
LIN {X 0,Y 58.393,Z 541.854,A -85,B 0,C 180,E1 -29414.319,E2 -29414.319} C_VEL
LIN {X 0,Y 53.399,Z 540.716,A -85,B 0,C 180,E1 -29403.214,E2 -29403.214} C_VEL
LIN {X 0,Y 50.735,Z 541.256,A -85,B 0,C 180,E1 -29405.445,E2 -29405.445} C_VEL
LIN {X 0,Y 47.471,Z 542.327,A -85,B 0,C 180,E1 -29412.777,E2 -29412.777} C_VEL
LIN {X 0,Y 45.139,Z 542.93,A -85,B 0,C 180,E1 -29421.043,E2 -29421.043} C_VEL
LIN {X 0,Y 43.959,Z 543.1,A -85,B 0,C 180,E1 -29430,E2 -29430} C_VEL
LIN {X 0,Y 45.114,Z 542.931,A -85,B 0,C 180,E1 -29438.962,E2 -29438.962} C_VEL
LIN {X 0,Y 47.469,Z 542.327,A -85,B 0,C 180,E1 -29447.224,E2 -29447.224} C_VEL
LIN {X 0,Y 50.734,Z 541.256,A -85,B 0,C 180,E1 -29454.555,E2 -29454.555} C_VEL
LIN {X 0,Y 53.283,Z 540.745,A -85,B 0,C 180,E1 -29456.653,E2 -29456.653} C_VEL
LIN {X 0,Y 54.24,Z 540.73,A -85,B 0,C 180,E1 -29456.117,E2 -29456.117} C_VEL
LIN {X 0,Y 54.861,Z 540.971,A -85,B 0,C 180,E1 -29453.984,E2 -29453.984} C_VEL
LIN {X 0,Y 54.948,Z 541.519,A -85,B 0,C 180,E1 -29449.788,E2 -29449.788} C_VEL
LIN {X 0,Y 55.089,Z 542.498,A -85,B 0,C 180,E1 -29440.018,E2 -29440.018} C_VEL
LIN {X 0,Y 56.892,Z 542.708,A -85,B 0,C 180,E1 -29435.73,E2 -29435.73} C_VEL
LIN {X 0,Y 57.465,Z 542.681,A -85,B 0,C 180,E1 -29435.018,E2 -29435.018} C_VEL
LIN {X 0,Y 62.646,Z 542.589,A -85,B 0,C 180,E1 -29430,E2 -29430} C_VEL
LIN {X 0,Y 54.163,Z 542.553,A -85,B 0,C 180,E1 -29420.807,E2 -29420.807} C_VEL
LIN {X 0,Y 52.202,Z 542.735,A -85,B 0,C 180,E1 -29422.263,E2 -29422.263} C_VEL
LIN {X 0,Y 51.082,Z 542.905,A -85,B 0,C 180,E1 -29430,E2 -29430} C_VEL
LIN {X 0,Y 52.18,Z 542.736,A -85,B 0,C 180,E1 -29437.74,E2 -29437.74} C_VEL
LIN {X 0,Y 54.103,Z 542.555,A -85,B 0,C 180,E1 -29439.197,E2 -29439.197} C_VEL
LIN {X 0,Y 57.465,Z 542.681,A -85,B 0,C 180,E1 -29435.018,E2 -29435.018} C_VEL
LIN {X 0,Y 58.84,Z 544.681,A -85,B 0,C 180,E1 -29433.554,E2 -29433.554} C_VEL
LIN {X 0,Y 58.84,Z 600,A -85,B 0,C 180,E1 -29433.554,E2 -29433.554} C_VEL
LIN {X 0,Y 58.84,Z 600,A -85,B 0,C 180,E1 -29433.554,E2 -29433.554}

QRS_NEXT_CUT()

QRS_NEXT()
QRS_HOME()

END
